(* IEC 61131-3 sources: SafePLC-Gen-Evaluation/PatchEvaluation-DEXPI-PDF, 2 files *)

(* ---- io_declarations.st ---- *)
(* ==================================================  *)
(* PLC I/O Variable Declarations — CODESYS 3.5  *)
(* Generated by SafePLC-Gen Multimodal  *)
(* ==================================================  *)

VAR_GLOBAL
    (* --- Analog Inputs ---  *)
    PI_4712.01_Raw               AT %IW0       : INT := 0;    (* PI-4712.01 — Pressure indicator on pump discharge  *)
    PICSA_4712.02_Raw            AT %IW2       : INT := 0;    (* PICSA-4712.02 — Pressure indicator controller switch ala  *)
    TICSA_4750.03_Raw            AT %IW4       : INT := 0;    (* TICSA-4750.03 — Temperature indicator controller switch   *)
    (* --- Analog Outputs ---  *)
    PV_71202_Out                 AT %QW0       : INT := 0;    (* PV-71202 — Pressure control valve with pneumatic di  *)
    TV_4750.03_Out               AT %QW2       : INT := 0;    (* TV-4750.03 — Temperature control valve with pneumatic  *)
    (* --- Digital Inputs ---  *)
    HS_4750.01                   AT %IX0.0     : BOOL := FALSE;    (* HS-4750.01 — Hand switch for manual operation  *)
    (* --- Digital Outputs ---  *)
    SV_104.01                    AT %QX0.0     : BOOL := FALSE;    (* SV-104.01 — Solenoid valve on vessel T4750 nozzle N5  *)
END_VAR

(* ---- generated_code.st ---- *)
(* Generated by SafePLC-Gen Multimodal — CODESYS 3.5 *)
(* IEC 61131-3 Structured Text *)
(* Date: 2026-04-15T12:55:26.932771 *)

PROGRAM Main
VAR
    (* AT-addressed I/O variables *)
    PI_4712_01_Raw               AT %IW0       : INT := 0;
    PICSA_4712_02_Raw            AT %IW2       : INT := 0;
    TICSA_4750_03_Raw            AT %IW4       : INT := 0;
    PV_71202_Out                 AT %QW0       : INT := 0;
    TV_4750_03_Out               AT %QW2       : INT := 0;
    HS_4750_01                   AT %IX0.0     : BOOL := FALSE;
    SV_104_01                    AT %QX0.0     : BOOL := FALSE;
END_VAR

VAR
    (* Internal variables *)
    FirstScan                    : BOOL := TRUE;

    (* Scaled process variables *)
    PI_4712_01_Scaled            : REAL := 0.0;
    PICSA_4712_02_Scaled         : REAL := 0.0;
    TICSA_4750_03_Scaled         : REAL := 0.0;
    HS_4750_01_Scaled            : REAL := 0.0;

    (* Alarm setpoints *)
    PI_4712_01_HH_SP             : REAL := 150.0;
    PI_4712_01_H_SP              : REAL := 120.0;
    PI_4712_01_L_SP              : REAL := 20.0;
    PI_4712_01_LL_SP             : REAL := 10.0;
    PI_4712_01_Deadband          : REAL := 5.0;

    PICSA_4712_02_HH_SP          : REAL := 160.0;
    PICSA_4712_02_H_SP           : REAL := 130.0;
    PICSA_4712_02_L_SP           : REAL := 25.0;
    PICSA_4712_02_LL_SP          : REAL := 15.0;
    PICSA_4712_02_Deadband       : REAL := 5.0;

    TICSA_4750_03_HH_SP          : REAL := 200.0;
    TICSA_4750_03_H_SP           : REAL := 180.0;
    TICSA_4750_03_L_SP           : REAL := 50.0;
    TICSA_4750_03_LL_SP          : REAL := 30.0;
    TICSA_4750_03_Deadband       : REAL := 10.0;

    HS_4750_01_HH_SP             : REAL := 1.5;
    HS_4750_01_H_SP              : REAL := 1.2;
    HS_4750_01_L_SP              : REAL := 0.3;
    HS_4750_01_LL_SP             : REAL := 0.1;
    HS_4750_01_Deadband          : REAL := 0.1;

    (* Alarm booleans *)
    PI_4712_01_HH                : BOOL := FALSE;
    PI_4712_01_H                 : BOOL := FALSE;
    PI_4712_01_L                 : BOOL := FALSE;
    PI_4712_01_LL                : BOOL := FALSE;

    PICSA_4712_02_HH             : BOOL := FALSE;
    PICSA_4712_02_H              : BOOL := FALSE;
    PICSA_4712_02_L              : BOOL := FALSE;
    PICSA_4712_02_LL             : BOOL := FALSE;

    TICSA_4750_03_HH             : BOOL := FALSE;
    TICSA_4750_03_H              : BOOL := FALSE;
    TICSA_4750_03_L              : BOOL := FALSE;
    TICSA_4750_03_LL             : BOOL := FALSE;

    HS_4750_01_HH                : BOOL := FALSE;
    HS_4750_01_H                 : BOOL := FALSE;
    HS_4750_01_L                 : BOOL := FALSE;
    HS_4750_01_LL                : BOOL := FALSE;

    (* Alarm latches *)
    PI_4712_01_HH_Latch          : SR := (S1 := FALSE, R := FALSE);
    PI_4712_01_LL_Latch          : SR := (S1 := FALSE, R := FALSE);
    PICSA_4712_02_HH_Latch       : SR := (S1 := FALSE, R := FALSE);
    PICSA_4712_02_LL_Latch       : SR := (S1 := FALSE, R := FALSE);
    TICSA_4750_03_HH_Latch       : SR := (S1 := FALSE, R := FALSE);
    TICSA_4750_03_LL_Latch       : SR := (S1 := FALSE, R := FALSE);
    HS_4750_01_HH_Latch          : SR := (S1 := FALSE, R := FALSE);
    HS_4750_01_LL_Latch          : SR := (S1 := FALSE, R := FALSE);

    (* Acknowledgement inputs *)
    PI_4712_01_HH_Ack            : BOOL := FALSE;
    PI_4712_01_LL_Ack            : BOOL := FALSE;
    PICSA_4712_02_HH_Ack         : BOOL := FALSE;
    PICSA_4712_02_LL_Ack         : BOOL := FALSE;
    TICSA_4750_03_HH_Ack         : BOOL := FALSE;
    TICSA_4750_03_LL_Ack         : BOOL := FALSE;
    HS_4750_01_HH_Ack            : BOOL := FALSE;
    HS_4750_01_LL_Ack            : BOOL := FALSE;

    (* Control variables *)
    PICSA_4712_02_SP             : REAL := 100.0;
    TICSA_4750_03_SP             : REAL := 150.0;

    (* PI Controller variables for PICSA-4712.02 *)
    PICSA_Error                  : REAL := 0.0;
    PICSA_Kp                     : REAL := 2.0;
    PICSA_Ki                     : REAL := 0.5;
    PICSA_Integral               : REAL := 0.0;
    PICSA_Output                 : REAL := 0.0;

    (* PI Controller variables for TICSA-4750.03 *)
    TICSA_Error                  : REAL := 0.0;
    TICSA_Kp                     : REAL := 1.5;
    TICSA_Ki                     : REAL := 0.3;
    TICSA_Integral               : REAL := 0.0;
    TICSA_Output                 : REAL := 0.0;

    (* System alarm aggregation *)
    System_Alarm                 : BOOL := FALSE;
END_VAR

(* First-scan initialization *)
IF FirstScan THEN
    (* Initialize safe states *)
    PV_71202_Out := 6554;
    TV_4750_03_Out := 6554;
    SV_104_01 := FALSE;

    (* Initialize alarm latches *)
    PI_4712_01_HH_Latch.S1 := FALSE;
    PI_4712_01_HH_Latch.R := FALSE;
    PI_4712_01_LL_Latch.S1 := FALSE;
    PI_4712_01_LL_Latch.R := FALSE;

    PICSA_4712_02_HH_Latch.S1 := FALSE;
    PICSA_4712_02_HH_Latch.R := FALSE;
    PICSA_4712_02_LL_Latch.S1 := FALSE;
    PICSA_4712_02_LL_Latch.R := FALSE;

    TICSA_4750_03_HH_Latch.S1 := FALSE;
    TICSA_4750_03_HH_Latch.R := FALSE;
    TICSA_4750_03_LL_Latch.S1 := FALSE;
    TICSA_4750_03_LL_Latch.R := FALSE;

    HS_4750_01_HH_Latch.S1 := FALSE;
    HS_4750_01_HH_Latch.R := FALSE;
    HS_4750_01_LL_Latch.S1 := FALSE;
    HS_4750_01_LL_Latch.R := FALSE;

    FirstScan := FALSE;
    RETURN;
END_IF;

(* Scale analog inputs *)
PI_4712_01_Scaled := ((INT_TO_REAL(PI_4712_01_Raw) - 6554.0) / (32767.0 - 6554.0)) * 200.0 + 0.0;
PICSA_4712_02_Scaled := ((INT_TO_REAL(PICSA_4712_02_Raw) - 6554.0) / (32767.0 - 6554.0)) * 200.0 + 0.0;
TICSA_4750_03_Scaled := ((INT_TO_REAL(TICSA_4750_03_Raw) - 6554.0) / (32767.0 - 6554.0)) * 300.0 + 0.0;

(* Scale digital input *)
IF HS_4750_01 THEN
    HS_4750_01_Scaled := 1.0;
ELSE
    HS_4750_01_Scaled := 0.0;
END_IF;

(* PI-4712.01 Four-level alarm logic *)
IF PI_4712_01_Scaled >= PI_4712_01_HH_SP THEN
    PI_4712_01_HH_Latch.S1 := TRUE;
ELSIF PI_4712_01_Scaled <= (PI_4712_01_HH_SP - PI_4712_01_Deadband) THEN
    PI_4712_01_HH_Latch.S1 := FALSE;
END_IF;

IF PI_4712_01_Scaled <= PI_4712_01_LL_SP THEN
    PI_4712_01_LL_Latch.S1 := TRUE;
ELSIF PI_4712_01_Scaled >= (PI_4712_01_LL_SP + PI_4712_01_Deadband) THEN
    PI_4712_01_LL_Latch.S1 := FALSE;
END_IF;

IF PI_4712_01_Scaled >= PI_4712_01_H_SP THEN
    PI_4712_01_H := TRUE;
ELSIF PI_4712_01_Scaled <= (PI_4712_01_H_SP - PI_4712_01_Deadband) THEN
    PI_4712_01_H := FALSE;
END_IF;

IF PI_4712_01_Scaled <= PI_4712_01_L_SP THEN
    PI_4712_01_L := TRUE;
ELSIF PI_4712_01_Scaled >= (PI_4712_01_L_SP + PI_4712_01_Deadband) THEN
    PI_4712_01_L := FALSE;
END_IF;

(* Acknowledge and reset HH/LL latches for PI-4712.01 *)
IF PI_4712_01_HH_Ack AND (PI_4712_01_Scaled <= (PI_4712_01_HH_SP - PI_4712_01_Deadband)) THEN
    PI_4712_01_HH_Latch.R := TRUE;
ELSE
    PI_4712_01_HH_Latch.R := FALSE;
END_IF;

IF PI_4712_01_LL_Ack AND (PI_4712_01_Scaled >= (PI_4712_01_LL_SP + PI_4712_01_Deadband)) THEN
    PI_4712_01_LL_Latch.R := TRUE;
ELSE
    PI_4712_01_LL_Latch.R := FALSE;
END_IF;

PI_4712_01_HH_Latch();
PI_4712_01_LL_Latch();

(* PICSA-4712.02 Four-level alarm logic *)
IF PICSA_4712_02_Scaled >= PICSA_4712_02_HH_SP THEN
    PICSA_4712_02_HH_Latch.S1 := TRUE;
ELSIF PICSA_4712_02_Scaled <= (PICSA_4712_02_HH_SP - PICSA_4712_02_Deadband) THEN
    PICSA_4712_02_HH_Latch.S1 := FALSE;
END_IF;

IF PICSA_4712_02_Scaled <= PICSA_4712_02_LL_SP THEN
    PICSA_4712_02_LL_Latch.S1 := TRUE;
ELSIF PICSA_4712_02_Scaled >= (PICSA_4712_02_LL_SP + PICSA_4712_02_Deadband) THEN
    PICSA_4712_02_LL_Latch.S1 := FALSE;
END_IF;

IF PICSA_4712_02_Scaled >= PICSA_4712_02_H_SP THEN
    PICSA_4712_02_H := TRUE;
ELSIF PICSA_4712_02_Scaled <= (PICSA_4712_02_H_SP - PICSA_4712_02_Deadband) THEN
    PICSA_4712_02_H := FALSE;
END_IF;

IF PICSA_4712_02_Scaled <= PICSA_4712_02_L_SP THEN
    PICSA_4712_02_L := TRUE;
ELSIF PICSA_4712_02_Scaled >= (PICSA_4712_02_L_SP + PICSA_4712_02_Deadband) THEN
    PICSA_4712_02_L := FALSE;
END_IF;

(* Acknowledge and reset HH/LL latches for PICSA-4712.02 *)
IF PICSA_4712_02_HH_Ack AND (PICSA_4712_02_Scaled <= (PICSA_4712_02_HH_SP - PICSA_4712_02_Deadband)) THEN
    PICSA_4712_02_HH_Latch.R := TRUE;
ELSE
    PICSA_4712_02_HH_Latch.R := FALSE;
END_IF;

IF PICSA_4712_02_LL_Ack AND (PICSA_4712_02_Scaled >= (PICSA_4712_02_LL_SP + PICSA_4712_02_Deadband)) THEN
    PICSA_4712_02_LL_Latch.R := TRUE;
ELSE
    PICSA_4712_02_LL_Latch.R := FALSE;
END_IF;

PICSA_4712_02_HH_Latch();
PICSA_4712_02_LL_Latch();

(* TICSA-4750.03 Four-level alarm logic *)
IF TICSA_4750_03_Scaled >= TICSA_4750_03_HH_SP THEN
    TICSA_4750_03_HH_Latch.S1 := TRUE;
ELSIF TICSA_4750_03_Scaled <= (TICSA_4750_03_HH_SP - TICSA_4750_03_Deadband) THEN
    TICSA_4750_03_HH_Latch.S1 := FALSE;
END_IF;

IF TICSA_4750_03_Scaled <= TICSA_4750_03_LL_SP THEN
    TICSA_4750_03_LL_Latch.S1 := TRUE;
ELSIF TICSA_4750_03_Scaled >= (TICSA_4750_03_LL_SP + TICSA_4750_03_Deadband) THEN
    TICSA_4750_03_LL_Latch.S1 := FALSE;
END_IF;

IF TICSA_4750_03_Scaled >= TICSA_4750_03_H_SP THEN
    TICSA_4750_03_H := TRUE;
ELSIF TICSA_4750_03_Scaled <= (TICSA_4750_03_H_SP - TICSA_4750_03_Deadband) THEN
    TICSA_4750_03_H := FALSE;
END_IF;

IF TICSA_4750_03_Scaled <= TICSA_4750_03_L_SP THEN
    TICSA_4750_03_L := TRUE;
ELSIF TICSA_4750_03_Scaled >= (TICSA_4750_03_L_SP + TICSA_4750_03_Deadband) THEN
    TICSA_4750_03_L := FALSE;
END_IF;

(* Acknowledge and reset HH/LL latches for TICSA-4750.03 *)
IF TICSA_4750_03_HH_Ack AND (TICSA_4750_03_Scaled <= (TICSA_4750_03_HH_SP - TICSA_4750_03_Deadband)) THEN
    TICSA_4750_03_HH_Latch.R := TRUE;
ELSE
    TICSA_4750_03_HH_Latch.R := FALSE;
END_IF;

IF TICSA_4750_03_LL_Ack AND (TICSA_4750_03_Scaled >= (TICSA_4750_03_LL_SP + TICSA_4750_03_Deadband)) THEN
    TICSA_4750_03_LL_Latch.R := TRUE;
ELSE
    TICSA_4750_03_LL_Latch.R := FALSE;
END_IF;

TICSA_4750_03_HH_Latch();
TICSA_4750_03_LL_Latch();

(* HS-4750.01 Four-level alarm logic *)
IF HS_4750_01_Scaled >= HS_4750_01_HH_SP THEN
    HS_4750_01_HH_Latch.S1 := TRUE;
ELSIF HS_4750_01_Scaled <= (HS_4750_01_HH_SP - HS_4750_01_Deadband) THEN
    HS_4750_01_HH_Latch.S1 := FALSE;
END_IF;

IF HS_4750_01_Scaled <= HS_4750_01_LL_SP THEN
    HS_4750_01_LL_Latch.S1 := TRUE;
ELSIF HS_4750_01_Scaled >= (HS_4750_01_LL_SP + HS_4750_01_Deadband) THEN
    HS_4750_01_LL_Latch.S1 := FALSE;
END_IF;

IF HS_4750_01_Scaled >= HS_4750_01_H_SP THEN
    HS_4750_01_H := TRUE;
ELSIF HS_4750_01_Scaled <= (HS_4750_01_H_SP - HS_4750_01_Deadband) THEN
    HS_4750_01_H := FALSE;
END_IF;

IF HS_4750_01_Scaled <= HS_4750_01_L_SP THEN
    HS_4750_01_L := TRUE;
ELSIF HS_4750_01_Scaled >= (HS_4750_01_L_SP + HS_4750_01_Deadband) THEN
    HS_4750_01_L := FALSE;
END_IF;

(* Acknowledge and reset HH/LL latches for HS-4750.01 *)
IF HS_4750_01_HH_Ack AND (HS_4750_01_Scaled <= (HS_4750_01_HH_SP - HS_4750_01_Deadband)) THEN
    HS_4750_01_HH_Latch.R := TRUE;
ELSE
    HS_4750_01_HH_Latch.R := FALSE;
END_IF;

IF HS_4750_01_LL_Ack AND (HS_4750_01_Scaled >= (HS_4750_01_LL_SP + HS_4750_01_Deadband)) THEN
    HS_4750_01_LL_Latch.R := TRUE;
ELSE
    HS_4750_01_LL_Latch.R := FALSE;
END_IF;

HS_4750_01_HH_Latch();
HS_4750_01_LL_Latch();

(* PICSA-4712.02 Pressure Control Loop - PI Controller *)
PICSA_Error := PICSA_4712_02_SP - PICSA_4712_02_Scaled;
PICSA_Integral := PICSA_Integral + (PICSA_Ki * PICSA_Error);

IF PICSA_Integral > 100.0 THEN
    PICSA_Integral := 100.0;
ELSIF PICSA_Integral < 0.0 THEN
    PICSA_Integral := 0.0;
END_IF;

PICSA_Output := (PICSA_Kp * PICSA_Error) + PICSA_Integral;

IF PICSA_Output > 100.0 THEN
    PICSA_Output := 100.0;
ELSIF PICSA_Output < 0.0 THEN
    PICSA_Output := 0.0;
END_IF;

(* TICSA-4750.03 Temperature Control Loop - PI Controller *)
TICSA_Error := TICSA_4750_03_SP - TICSA_4750_03_Scaled;
TICSA_Integral := TICSA_Integral + (TICSA_Ki * TICSA_Error);

IF TICSA_Integral > 100.0 THEN
    TICSA_Integral := 100.0;
ELSIF TICSA_Integral < 0.0 THEN
    TICSA_Integral := 0.0;
END_IF;

TICSA_Output := (TICSA_Kp * TICSA_Error) + TICSA_Integral;

IF TICSA_Output > 100.0 THEN
    TICSA_Output := 100.0;
ELSIF TICSA_Output < 0.0 THEN
    TICSA_Output := 0.0;
END_IF;

(* Output scaling and assignments *)
PV_71202_Out := REAL_TO_INT(6554.0 + (PICSA_Output / 100.0) * (32767.0 - 6554.0));
TV_4750_03_Out := REAL_TO_INT(6554.0 + (TICSA_Output / 100.0) * (32767.0 - 6554.0));

(* Solenoid valve control based on hand switch *)
SV_104_01 := HS_4750_01;

(* Aggregate all alarm states for SCADA/HMI *)
System_Alarm :=
    PI_4712_01_HH_Latch.Q1 OR PI_4712_01_LL_Latch.Q1 OR
    PI_4712_01_H           OR PI_4712_01_L            OR
    PICSA_4712_02_HH_Latch.Q1 OR PICSA_4712_02_LL_Latch.Q1 OR
    PICSA_4712_02_H           OR PICSA_4712_02_L            OR
    TICSA_4750_03_HH_Latch.Q1 OR TICSA_4750_03_LL_Latch.Q1 OR
    TICSA_4750_03_H           OR TICSA_4750_03_L            OR
    HS_4750_01_HH_Latch.Q1    OR HS_4750_01_LL_Latch.Q1    OR
    HS_4750_01_H              OR HS_4750_01_L;

END_PROGRAM
